// TIA Portal V18 export
DATA_BLOCK "Temp"   // DB167
{ S7_Optimized_Access := 'TRUE' }
VERSION : 0.1
// stored: AutoNumber true, DBAccessibleFromOPCUA true, IsOnlyStoredInLoadMemory false, IsRetainMemResEnabled false, IsWriteProtectedInAS false, MemoryReserve 100
   VAR
      bit1 : Bool;
      bit2 : Bool;
      bit3 : Bool;
      bit4 : Bool;
      bit5 : Bool;
      bit6 : Bool;
      bit7 : Bool;
      bit8 : Bool;
      bit9 : Bool;
      bit10 : Bool;
      bit11 : Bool;
      bit12 : Bool;
      bit13 : Bool;
      bit14 : Bool;
      bit15 : Bool;
      bit16 : Bool;
      bit17 : Bool;
      bit18 : Bool;
      bit19 : Bool;
      bit20 : Bool;
      bit21 : Bool;
      bit22 : Bool;
      bit23 : Bool;
      bit24 : Bool;
      bit25 : Bool;
      bit26 : Bool;
      bit27 : Bool;
      temp : Int;
      temp_1 : Int;
      temp_2 : Int;
      temp_3 : Array[0..30] of Bool;
   END_VAR
   VAR RETAIN
      Snuffback_ONdelay_A : Time := T#5MS;
      Snuffback_OFFdelay_A : Time := T#5MS;
      Snuffback_Ondelay_B : Time := T#1S;
      Snuffback_OFFdelay_B : Time := T#1S;
   END_VAR
   VAR
      Snuffback_vol_dispensedA { ExternalAccessible := 'False'; ExternalVisible := 'False'; ExternalWritable := 'False'} : Real;
      Snuffback_vol_dispensedB { ExternalAccessible := 'False'; ExternalVisible := 'False'; ExternalWritable := 'False'} : Real;
      Metering_time_inSec { ExternalAccessible := 'False'; ExternalVisible := 'False'; ExternalWritable := 'False'} : Time;
   END_VAR
   VAR RETAIN
      Language_selection : Int;
   END_VAR
   VAR
      temp_4 : Array[0..10] of Bool;
      ratiocheck_temp : Array[0..10] of Bool;
   END_VAR
BEGIN
END_DATA_BLOCK
